FUNCTION_BLOCK SampleComponentTests EXTENDS TcoCore._internals_TcoContext
VAR
	_sut : TcoIoBeckhoff.SampleComponent(THIS^);
END_VAR

{attribute 'TcRpcEnable'}
METHOD INTERNAL AddTwoNumbersTest : INT
VAR_INPUT
	NumberOne : INT;
	NumberTwo : INT;
END_VAR
AddTwoNumbersTest := _sut.AddTwoNumbers(NumberOne, NumberTwo);
END_METHOD

METHOD PROTECTED Main
END_METHOD

{attribute 'TcRpcEnable'}
METHOD INTERNAL WaitForModuloTest : BOOL
VAR_INPUT
	Modulo : INT;
END_VAR
WaitForModuloTest := _sut.WaitForModulo(Modulo);
END_METHOD

END_FUNCTION_BLOCK

(* stored: Version 1.1.0.1, ProductVersion 3.1.4024.9
   POU SampleComponentTests: Id {59d24b2c-148b-081d-164b-e04a36fdd44a}, SpecialFunc None
   Method AddTwoNumbersTest: Id {9c2bb0cc-4b78-00fe-3a26-c17460dad23a}
   Method Main: Id {f9c63a21-8864-04ed-1cb7-fda475bab4cf}
   Method WaitForModuloTest: Id {1620f468-f32b-0f25-0b1d-f21773abde6d} *)
